SUBAPPLICATION Uebung_006a3 (* SR und T-Flip-Flop mit 3x IE *)
  (* Standard: 61499-2; Description: Copyright (c) 2023 Meisterschulen am Ostbahnhof This program and the accompanying materials are made available under the terms of the Eclipse Public License 2.0 which is available at https://www.eclipse.org/legal/epl-2.0/ SPDX-License-Identifier: EPL-2.0 *)
  (* Version 1.0, 2023-10-23, Franz Höpfinger, Meisterschulen am Ostbahnhof *)
  PACKAGE Uebungen;
  IMPORT logiBUS::io::DI::logiBUS_DI::Input_I1;
  IMPORT logiBUS::io::DI::logiBUS_DI::Input_I2;
  IMPORT logiBUS::io::DI::logiBUS_DI::Input_I3;
  IMPORT logiBUS::io::DI::logiBUS_DI_Events::BUTTON_SINGLE_CLICK;
  IMPORT logiBUS::io::DQ::logiBUS_DO::Output_Q1;
  IMPORT logiBUS::io::DQ::logiBUS_DO::Output_Q2;
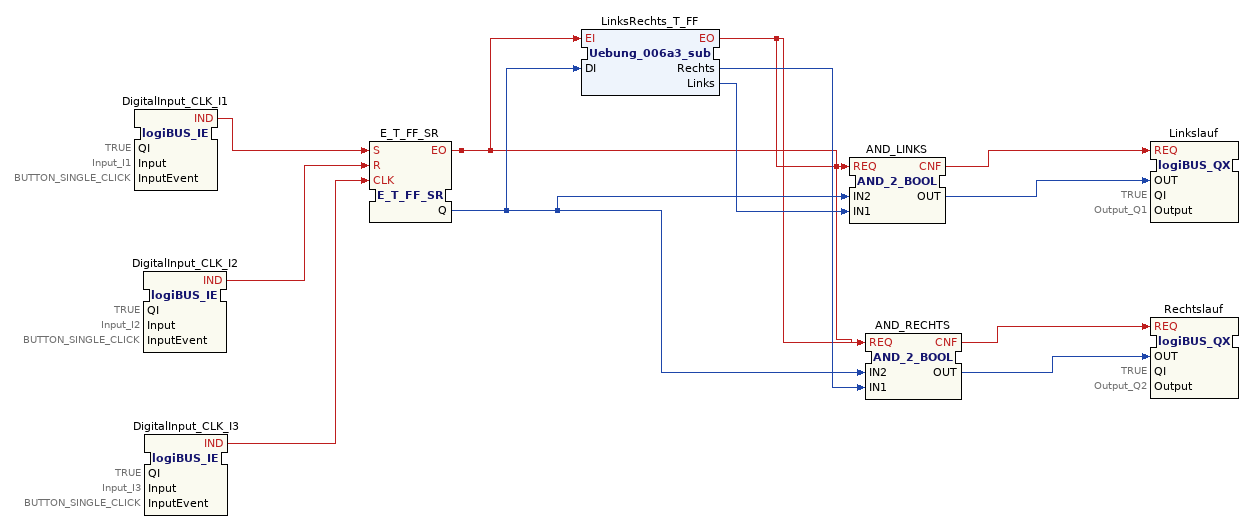
  FBS
    DigitalInput_CLK_I1 : logiBUS::io::DI::logiBUS_IE(QI := TRUE, Input := Input_I1, InputEvent := BUTTON_SINGLE_CLICK);
    DigitalInput_CLK_I2 : logiBUS::io::DI::logiBUS_IE(QI := TRUE, Input := Input_I2, InputEvent := BUTTON_SINGLE_CLICK);
    E_T_FF_SR : iec61499::events::E_T_FF_SR;
    DigitalInput_CLK_I3 : logiBUS::io::DI::logiBUS_IE(QI := TRUE, Input := Input_I3, InputEvent := BUTTON_SINGLE_CLICK);
    AND_LINKS : iec61131::bitwiseOperators::AND_2_BOOL;
    Rechtslauf : logiBUS::io::DQ::logiBUS_QX(QI := TRUE, Output := Output_Q2);
    Linkslauf : logiBUS::io::DQ::logiBUS_QX(QI := TRUE, Output := Output_Q1);
    AND_RECHTS : iec61131::bitwiseOperators::AND_2_BOOL;
  END_FBS
  SUBAPPS
    LinksRechts_T_FF : Uebungen::Uebung_006a3_sub;
  END_SUBAPPS
  EVENT_CONNECTIONS
    DigitalInput_CLK_I1.IND TO E_T_FF_SR.S;
    DigitalInput_CLK_I2.IND TO E_T_FF_SR.R;
    DigitalInput_CLK_I3.IND TO E_T_FF_SR.CLK;
    AND_RECHTS.CNF TO Rechtslauf.REQ;
    AND_LINKS.CNF TO Linkslauf.REQ;
    E_T_FF_SR.EO TO LinksRechts_T_FF.EI;
    LinksRechts_T_FF.EO TO AND_LINKS.REQ;
    LinksRechts_T_FF.EO TO AND_RECHTS.REQ;
    E_T_FF_SR.EO TO AND_LINKS.REQ;
    E_T_FF_SR.EO TO AND_RECHTS.REQ;
  END_CONNECTIONS
  DATA_CONNECTIONS
    AND_LINKS.OUT TO Linkslauf.OUT;
    E_T_FF_SR.Q TO AND_RECHTS.IN2;
    AND_RECHTS.OUT TO Rechtslauf.OUT;
    E_T_FF_SR.Q TO AND_LINKS.IN2;
    LinksRechts_T_FF.Rechts TO AND_RECHTS.IN1;
    E_T_FF_SR.Q TO LinksRechts_T_FF.DI;
    LinksRechts_T_FF.Links TO AND_LINKS.IN1;
  END_CONNECTIONS
END_SUBAPPLICATION
